// TIA Portal V21 export
// export: ExportSetting WithDefaults
FUNCTION_BLOCK "Ref_TonSR_Verify"   // FB103, LAD
{ S7_Optimized_Access := 'TRUE' }
VERSION : 0.1
// stored: AutoNumber true, IsIECCheckEnabled true, SetENOAutomatically false, UDAEnableTagReadback false
   VAR_INPUT
      Start : Bool;
      Trig : Bool;
      Rst : Bool;
   END_VAR
   VAR_OUTPUT
      Done : Bool;
      Latch : Bool;
   END_VAR
   VAR
      "Timer" : TON_TIME;
   END_VAR
BEGIN

REGION Network 1
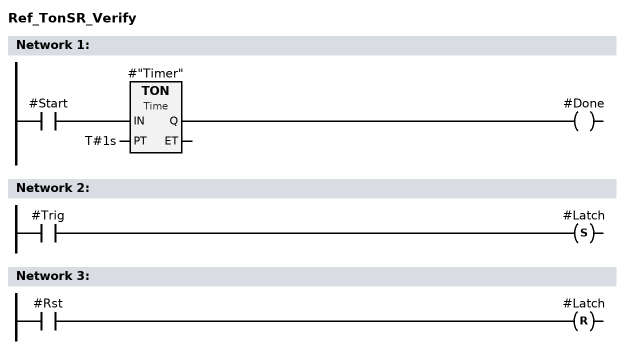
   RUNG wire#powerrail
      Contact( #Start )
      { S7_Templates := "time_type := Time" } #"Timer".TON(pt := T#1s, et =>)
      Coil( #Done )
   END_RUNG
   // the same network as SCL:
   #"Timer"(IN := #Start, PT := T#1s);   // TON
   #Done := #"Timer".Q;
END_REGION

REGION Network 2
   RUNG wire#powerrail
      Contact( #Trig )
      S_Coil( #Latch )
   END_RUNG
   // the same network as SCL:
   IF #Trig THEN #Latch := TRUE; END_IF;
END_REGION

REGION Network 3
   RUNG wire#powerrail
      Contact( #Rst )
      R_Coil( #Latch )
   END_RUNG
   // the same network as SCL:
   IF #Rst THEN #Latch := FALSE; END_IF;
END_REGION
END_FUNCTION_BLOCK
